{attribute 'GeneratedUsingTerminal: ER1518-0002-0018'}
{attribute addProperty BoxType "ER1518-0002-0018"}
{attribute addProperty Id "StatusAT %I*Status_57491DF17Counter_valueAT %I*UDINT4"}
{attribute addProperty CRC "4279287100"}
{attribute addProperty Size "11"}
TYPE CNT_Input_Channel_FF10BD3C :
STRUCT
	{attribute addProperty Name "Status"}
	Status AT %I* : Status_57491DF1;
	{attribute addProperty Name "Counter_value"}
	Counter_value AT %I* : UDINT;
END_STRUCT
END_TYPE

(* stored: Version 1.2.0.0, ProductVersion 3.1.4024.9
   DUT CNT_Input_Channel_FF10BD3C: Id {9c06aad3-8d7a-494e-b7b7-1311ba961f9b} *)
